FUNCTION_BLOCK TAssertionListenerMock IMPLEMENTS IAssertionListener
VAR
    {attribute 'instance-path'} 
    {attribute 'no_init'}
    _TestName : T_MaxString; // Automatically initialised with the full name of the instance
    _AssertionFailed  : BOOL;
    _AssertionMessage : T_MaxString;
    _ExpectedAsString : T_MaxString;
    _ActualAsString   : T_MaxString;
END_VAR

PROPERTY ActualAsString : T_MaxString
GET
ActualAsString := _ActualAsString;
END_GET
SET
_ActualAsString := ActualAsString;
END_SET
END_PROPERTY

PROPERTY AssertionFailed : BOOL
GET
AssertionFailed := _AssertionFailed;
END_GET
SET
_AssertionFailed := AssertionFailed;
END_SET
END_PROPERTY

PROPERTY AssertionMessage : T_MaxString
GET
AssertionMessage := _AssertionMessage;
END_GET
SET
_AssertionMessage := AssertionMessage;
END_SET
END_PROPERTY

PROPERTY ExpectedAsString : T_MaxString
GET
ExpectedAsString := _ExpectedAsString;
END_GET
SET
_ExpectedAsString := ExpectedAsString;
END_SET
END_PROPERTY

METHOD OnAssertionFailed
VAR_INPUT
    AssertionMessage : T_MaxString;
    ExpectedAsString : T_MaxString;
    ActualAsString   : T_MaxString;
END_VAR
_AssertionFailed   := TRUE;
_AssertionMessage  := AssertionMessage;
_ExpectedAsString := ExpectedAsString;
_ActualAsString := ActualAsString;
END_METHOD

PROPERTY TestName : Tc2_System.T_MaxString
GET
TestName := _TestName;
END_GET
END_PROPERTY

END_FUNCTION_BLOCK

(* stored: Version 1.1.0.1, ProductVersion 3.1.4024.4
   POU TAssertionListenerMock: Id {ee93dd0b-67fe-45ad-ace0-2b0e0c9dee67}, SpecialFunc None
   Property ActualAsString: Id {c1cce4b8-2ad7-4260-a30c-42c9cfb3867c}
   Get Get: Id {c15f9fb9-fe7e-48ba-bcc3-1ad21cfbb84c}
   Set Set: Id {39495475-1c93-499a-92db-f4cbcc366715}
   Property AssertionFailed: Id {8877a547-33cb-47d7-baea-06c57dc3053d}
   Get Get: Id {fe4188fc-a128-4ef2-8667-c6e21445f7de}
   Set Set: Id {de257556-911c-4385-8e9d-cbaa9bb3502f}
   Property AssertionMessage: Id {2389e857-4bcb-4ea5-b2a3-969d29fbf6fa}
   Get Get: Id {e66eef02-5cbe-4381-a588-ea502a1598d1}
   Set Set: Id {b34472cd-3976-468b-898b-a13818876f5d}
   Property ExpectedAsString: Id {ad944bb0-d188-43f0-b8fb-3322e444535b}
   Get Get: Id {d7ab7b51-8787-483c-9bd2-fc32abd1237d}
   Set Set: Id {80e4777c-89c3-479f-a122-f779f83bc93a}
   Method OnAssertionFailed: Id {33a7986a-d29d-4499-9710-f64583918101}
   Property TestName: Id {4df2820b-acf9-463d-a62d-b441799ed9a6}
   Get Get: Id {965b97f0-d6de-46bc-9c27-21a8645aa650} *)
